# B&R Automation Studio project Intro_5_3_2020
Automation Studio 4.7.2.98

## Configuration Config1

CPU X20CP1584, AutomationRuntime C4.72, Build 4.1.2, Vc V4.72.0

### Task classes (Cpu.sw)
```
Cyclic#4:
  Program <- Program.prg
Binaries: udbdef, FWRules, TCData, iomap, ashwac, Role, sysconf, arconfig, asfw, User, ashwd
Libraries: standard
```

### Hardware
```
X20CP1584 : X20CP1584 v1.6.0.0
  Connector IF2:
    ActivateDevice = 1
  ConfigurationID = Intro_5_3_2020_Config1
  Simulation = 1
```

## Logical view

### Program Logical/Program (ANSIC)

#### Variables.var
```iecst
VAR
	Time_on : TON;
	OUT : BOOL;
	IN2 : BOOL;
	IN1 : BOOL;
	ON_Del : TIME;
END_VAR
```

#### Cyclic.c
```c
#include <bur/plctypes.h>
#include <standard.h>
#ifdef _DEFAULT_INCLUDES
	#include <AsDefault.h>
#endif

void _CYCLIC ProgramCyclic(void)
{
	Time_on.IN = IN1;
	OUT = Time_on.Q;
	TON(&Time_on);
}
```

#### Init.c
```c
#include <bur/plctypes.h>

#ifdef _DEFAULT_INCLUDES
	#include <AsDefault.h>
#endif

void _INIT ProgramInit(void)
{
	IN1 = 0;
	IN2 = 0;
	OUT = 1;
	ON_Del = 1000;
	Time_on.PT = ON_Del;
}
```

Listed in the project but not available here: Logical/Global.typ, Logical/Global.var, Logical/Libraries
